SYSTEM Distributed_Control_System_OPCUA_4Diac
  (* Version 1.0, Author, Eclipse 4diac *)
  APPLICATION Distributed_Control_System_OPCUA_4DiacApp
    FBS
      HMI_COME_TO_ME : HMI_COME_TO_ME;
      EMERGENCY_STOP : RADIO_BOOL(QI := 1, LABEL1 := Start, LABEL0 := Emergency STOP, IN := 0);
      INPUT_BOX : IN_ANY(QI := 1, W := 20, TYPE := INT);
      COME_TO_ME : RADIO_BOOL(QI := 1, LABEL1 := Come to me, LABEL0 := STOP, IN := 0);
      FOLLOW_ME : RADIO_BOOL(QI := 1, LABEL1 := Follow me, LABEL0 := STOP, IN := 0);
      FOLLOW_MACHINE : RADIO_BOOL(QI := 1, LABEL1 := Follow machine, LABEL0 := STOP, IN := 0);
      INT2INT : INT2INT;
      HMI_FOLLOW_ME : HMI_FOLLOW_ME;
      HMI_FOLLOW_MACHINE : HMI_FOLLOW_MACHINE;
      CRANE2_COME_TO_ME : CRANE2_COME_TO_ME;
      CRANE1_COME_TO_ME : CRANE1_COME_TO_ME;
      CRANE2_FOLLOW_ME : CRANE2_FOLLOW_ME;
      CRANE1_FOLLOW_MACHINE : CRANE1_FOLLOW_MACHINE;
      CRANE2_FOLLOW_MACHINE : CRANE2_FOLLOW_MACHINE;
      MASTER_SLAVE : RADIO_BOOL(QI := 1, LABEL1 := Activate Bridge, LABEL0 := Stop, IN := 0);
      ACTIVATE_TROLLEY : RADIO_BOOL(QI := 1, LABEL1 := Activate Trolley, LABEL0 := Stop, IN := 0);
      ACTIVATE_HOOK : RADIO_BOOL(QI := 1, LABEL1 := Hook Up, LABEL0 := Stop, IN := 0);
      CRANE_NR : RADIO_BOOL(QI := 1, LABEL1 := Select Crane Nr, LABEL0 := No, IN := 0);
      HOOK_UP_DOWN : RADIO_BOOL(QI := 1, LABEL1 := Hook Down, LABEL0 := Stop, IN := 0);
      SENSORS_ACTUATORS_2 : SENSORS_ACTUATORS;
      SENSORS_ACTUATORS_1 : SENSORS_ACTUATORS;
      CHOOSE_X : RADIO_BOOL(QI := 1, LABEL1 := Choose X, LABEL0 := No, IN := 0);
      CHOOSE_Y : RADIO_BOOL(QI := 1, LABEL1 := Choose Y, LABEL0 := No, IN := 0);
      BOOL2BOOL : BOOL2BOOL;
      BOOL2BOOL_1 : BOOL2BOOL;
      CRANE_1 : CLIENT_6_0(QI := 1, ID := opc_ua[opc.tcp://%CRANE1_IP%:4840#/Objects/1:CRANE1/SERVER1]);
      CEANE_2 : CLIENT_6_0(QI := 1, ID := opc_ua[opc.tcp://%CRANE2_IP%:4840#/Objects/1:CRANE2/SERVER2]);
      TYPE_CONVERTER : TYPE_CONVERTER_1I_11B;
      SERVER1 : SERVER_0_6(QI := 1, ID := opc_ua[/Objects/1:CRANE1]);
      FUNCTIONALITY_CONTROLLER : FUNCTIONALITY_CONTROLLER;
      CRANE_SELECTOR : CRANE_SELECTOR;
      FME_FMA_DECIDER : FME_FMA_DECIDER;
      CRANE1_FOLLOW_ME : CRANE1_FOLLOW_ME;
      SUBSCRIBE_10_2 : SUBSCRIBE_10(QI := 1, ID := 239.0.0.2:61497);
      SERVER2 : SERVER_0_6(QI := 1, ID := opc_ua[/Objects/1:CRANE2]);
      PUBLISH_10 : PUBLISH_10(QI := 1, ID := 239.0.0.2:61497);
      SUB1 : SUBSCRIBE_10(QI := 1, ID := 239.0.0.2:61497);
      PUBLISH_12 : PUBLISH_12(QI := 1, ID := 239.0.0.1:61496);
      SUBSCRIBE_12 : SUBSCRIBE_12(QI := 1, ID := 239.0.0.1:61496);
      START_STOP_CONTROLLER_1 : START_STOP_CONTROLLER;
      START_STOP_CONTROLLER_2 : START_STOP_CONTROLLER;
      REQUEST : DISPLAY_LOCAL_TIME;
      RESPONSE : DISPLAY_LOCAL_TIME;
      PERMITTER_2 : PERMITTER;
      PERMITTER_1 : PERMITTER;
      BOOL2BOOL_2 : BOOL2BOOL;
      BOOL2BOOL_3 : BOOL2BOOL;
    END_FBS
    EVENT_CONNECTIONS
      INPUT_BOX.IND TO INT2INT.REQ;
      EMERGENCY_STOP.INITO TO INPUT_BOX.INIT;
      INPUT_BOX.INITO TO COME_TO_ME.INIT;
      COME_TO_ME.INITO TO FOLLOW_ME.INIT;
      FOLLOW_ME.INITO TO FOLLOW_MACHINE.INIT;
      MASTER_SLAVE.INITO TO ACTIVATE_TROLLEY.INIT;
      ACTIVATE_TROLLEY.INITO TO ACTIVATE_HOOK.INIT;
      CRANE2_COME_TO_ME.CNF TO SENSORS_ACTUATORS_2.REQ;
      CRANE1_COME_TO_ME.CNF TO SENSORS_ACTUATORS_1.REQ;
      CRANE1_FOLLOW_MACHINE.CNF TO SENSORS_ACTUATORS_1.REQ;
      CHOOSE_X.INITO TO CHOOSE_Y.INIT;
      HOOK_UP_DOWN.INITO TO CHOOSE_X.INIT;
      CHOOSE_Y.IND TO BOOL2BOOL_1.REQ;
      CHOOSE_X.IND TO BOOL2BOOL.REQ;
      FOLLOW_MACHINE.INITO TO CRANE_NR.INIT;
      CRANE_NR.INITO TO MASTER_SLAVE.INIT;
      ACTIVATE_HOOK.INITO TO HOOK_UP_DOWN.INIT;
      SERVER1.IND TO CRANE1_COME_TO_ME.REQ;
      SERVER1.IND TO CRANE1_FOLLOW_MACHINE.REQ;
      SERVER1.INITO TO SENSORS_ACTUATORS_1.INIT;
      TYPE_CONVERTER.CNF TO HMI_COME_TO_ME.REQ;
      TYPE_CONVERTER.CNF TO HMI_FOLLOW_ME.REQ;
      TYPE_CONVERTER.CNF TO HMI_FOLLOW_MACHINE.REQ;
      TYPE_CONVERTER.CNF TO FUNCTIONALITY_CONTROLLER.TRIGGER;
      FUNCTIONALITY_CONTROLLER.CTM_OUT TO HMI_COME_TO_ME.TRIGGER_IN;
      SERVER1.IND TO SERVER1.RSP;
      CRANE2_FOLLOW_ME.CNF TO SENSORS_ACTUATORS_2.REQ;
      CRANE2_FOLLOW_MACHINE.CNF TO SENSORS_ACTUATORS_2.REQ;
      FUNCTIONALITY_CONTROLLER.FME_OUT TO HMI_FOLLOW_ME.TRIGGER_IN;
      FUNCTIONALITY_CONTROLLER.FMA_OUT TO HMI_FOLLOW_MACHINE.TRIGGER_IN;
      HMI_COME_TO_ME.TRIGGER_OUT TO CRANE_SELECTOR.CTM;
      HMI_FOLLOW_ME.TRIGGER_OUT TO CRANE_SELECTOR.FME;
      TYPE_CONVERTER.CNF TO CRANE_SELECTOR.REQ;
      HMI_FOLLOW_MACHINE.TRIGGER_OUT TO CRANE_SELECTOR.FMA;
      SENSORS_ACTUATORS_1.S_A_E TO CRANE1_COME_TO_ME.MPS_E;
      SENSORS_ACTUATORS_1.S_A_E TO CRANE1_FOLLOW_MACHINE.MPS_E;
      SENSORS_ACTUATORS_2.S_A_E TO CRANE2_FOLLOW_ME.MPS_E;
      SENSORS_ACTUATORS_2.S_A_E TO CRANE2_COME_TO_ME.MPS_E;
      SENSORS_ACTUATORS_2.S_A_E TO CRANE2_FOLLOW_MACHINE.MPS_E;
      HMI_COME_TO_ME.UPDATER_OUT TO HMI_FOLLOW_ME.REQ;
      HMI_COME_TO_ME.UPDATER_OUT TO HMI_FOLLOW_MACHINE.REQ;
      HMI_FOLLOW_ME.TRIGGER_OUT TO FME_FMA_DECIDER.FME_TRIGGER;
      HMI_FOLLOW_MACHINE.TRIGGER_OUT TO FME_FMA_DECIDER.FMA_TRIGGER;
      FME_FMA_DECIDER.TRIGGER TO HMI_COME_TO_ME.UPDATER_IN;
      CRANE1_FOLLOW_ME.CNF TO SENSORS_ACTUATORS_1.REQ;
      SENSORS_ACTUATORS_1.S_A_E TO CRANE1_FOLLOW_ME.MPS_E;
      SERVER1.IND TO CRANE1_FOLLOW_ME.REQ;
      SERVER2.INITO TO SUBSCRIBE_10_2.INIT;
      TYPE_CONVERTER.CNF TO PUBLISH_10.REQ;
      SERVER1.INITO TO SUB1.INIT;
      SUB1.IND TO CRANE1_COME_TO_ME.REQ;
      SUB1.IND TO CRANE1_FOLLOW_ME.REQ;
      SUB1.IND TO SENSORS_ACTUATORS_1.REQ;
      PUBLISH_12.INITO TO EMERGENCY_STOP.INIT;
      EMERGENCY_STOP.IND TO PUBLISH_12.REQ;
      INT2INT.CNF TO PUBLISH_12.REQ;
      COME_TO_ME.IND TO PUBLISH_12.REQ;
      FOLLOW_ME.IND TO PUBLISH_12.REQ;
      FOLLOW_MACHINE.IND TO PUBLISH_12.REQ;
      CRANE_NR.IND TO PUBLISH_12.REQ;
      MASTER_SLAVE.IND TO PUBLISH_12.REQ;
      ACTIVATE_TROLLEY.IND TO PUBLISH_12.REQ;
      ACTIVATE_HOOK.IND TO PUBLISH_12.REQ;
      HOOK_UP_DOWN.IND TO PUBLISH_12.REQ;
      BOOL2BOOL.CNF TO PUBLISH_12.REQ;
      BOOL2BOOL_1.CNF TO PUBLISH_12.REQ;
      SUBSCRIBE_12.IND TO TYPE_CONVERTER.REQ;
      SUBSCRIBE_12.INITO TO PUBLISH_10.INIT;
      SUBSCRIBE_12.INITO TO CRANE_1.INIT;
      SUBSCRIBE_12.INITO TO CEANE_2.INIT;
      SUB1.IND TO START_STOP_CONTROLLER_1.REQ;
      SUB1.INITO TO START_STOP_CONTROLLER_1.INIT;
      START_STOP_CONTROLLER_1.CNF TO CRANE1_FOLLOW_ME.REQ;
      START_STOP_CONTROLLER_1.CNF TO CRANE1_COME_TO_ME.REQ;
      START_STOP_CONTROLLER_2.CNF TO CRANE2_COME_TO_ME.REQ;
      START_STOP_CONTROLLER_2.CNF TO CRANE2_FOLLOW_MACHINE.REQ;
      START_STOP_CONTROLLER_2.CNF TO CRANE2_FOLLOW_ME.REQ;
      START_STOP_CONTROLLER_1.CNF TO CRANE1_FOLLOW_MACHINE.REQ;
      SUB1.IND TO CRANE1_FOLLOW_MACHINE.REQ;
      SERVER2.IND TO CRANE2_COME_TO_ME.REQ;
      SERVER2.IND TO CRANE2_FOLLOW_ME.REQ;
      SERVER2.IND TO CRANE2_FOLLOW_MACHINE.REQ;
      SERVER2.IND TO SERVER2.RSP;
      SUBSCRIBE_10_2.INITO TO SENSORS_ACTUATORS_2.INIT;
      SUBSCRIBE_10_2.INITO TO START_STOP_CONTROLLER_2.INIT;
      SUBSCRIBE_10_2.IND TO CRANE2_COME_TO_ME.REQ;
      SUBSCRIBE_10_2.IND TO CRANE2_FOLLOW_ME.REQ;
      SUBSCRIBE_10_2.IND TO CRANE2_FOLLOW_MACHINE.REQ;
      SUBSCRIBE_10_2.IND TO SENSORS_ACTUATORS_2.REQ;
      SUBSCRIBE_10_2.IND TO START_STOP_CONTROLLER_2.REQ;
      CRANE_SELECTOR.C2 TO CEANE_2.REQ;
      CRANE_SELECTOR.C1 TO CRANE_1.REQ;
      CRANE_1.CNF TO RESPONSE.REQ;
      CEANE_2.CNF TO RESPONSE.REQ;
      CRANE_SELECTOR.C1 TO REQUEST.REQ;
      CRANE_SELECTOR.C2 TO REQUEST.REQ;
      START_STOP_CONTROLLER_1.CNF TO PERMITTER_1.REQ;
      SENSORS_ACTUATORS_1.S_A_E TO PERMITTER_1.TRIGGER_IN;
      PERMITTER_1.TRIGGER_OUT TO CRANE1_FOLLOW_MACHINE.REQ;
      START_STOP_CONTROLLER_2.CNF TO PERMITTER_2.REQ;
      SENSORS_ACTUATORS_2.S_A_E TO PERMITTER_2.TRIGGER_IN;
      PERMITTER_2.TRIGGER_OUT TO CRANE2_FOLLOW_MACHINE.REQ;
    END_CONNECTIONS
    DATA_CONNECTIONS
      INPUT_BOX.OUT TO INT2INT.IN;
      SENSORS_ACTUATORS_2.CRANE_DIS_S TO CRANE2_COME_TO_ME.CRANE_DIS_S;
      SENSORS_ACTUATORS_1.CRANE_DIS_S TO CRANE1_COME_TO_ME.CRANE_DIS_S;
      SENSORS_ACTUATORS_1.CRANE_DIS_S TO CRANE1_FOLLOW_MACHINE.CRANE_DIS_S;
      SENSORS_ACTUATORS_2.CRANE_DIS_S TO CRANE2_FOLLOW_ME.CRANE_DIS_S;
      SENSORS_ACTUATORS_2.CRANE_DIS_S TO CRANE2_FOLLOW_MACHINE.CRANE_DIS_S;
      CHOOSE_Y.OUT TO BOOL2BOOL_1.IN;
      CHOOSE_X.OUT TO BOOL2BOOL.IN;
      TYPE_CONVERTER.BOOL11OUT TO HMI_COME_TO_ME.Choose_X;
      TYPE_CONVERTER.BOOL12OUT TO HMI_COME_TO_ME.Choose_Y;
      TYPE_CONVERTER.BOOL11OUT TO HMI_FOLLOW_ME.Choose_X;
      TYPE_CONVERTER.BOOL12OUT TO HMI_FOLLOW_ME.Choose_Y;
      TYPE_CONVERTER.BOOL12OUT TO HMI_FOLLOW_MACHINE.Choose_Y;
      HMI_COME_TO_ME.Output_X TO CRANE_SELECTOR.CTM_X_I;
      HMI_COME_TO_ME.Output_Y TO CRANE_SELECTOR.CTM_Y_I;
      HMI_FOLLOW_ME.Output_X TO CRANE_SELECTOR.FME_X_I;
      HMI_FOLLOW_ME.Output_Y TO CRANE_SELECTOR.FME_Y_I;
      HMI_FOLLOW_MACHINE.Output_X TO CRANE_SELECTOR.FMA_X_I;
      HMI_FOLLOW_MACHINE.Output_Y TO CRANE_SELECTOR.FMA_Y_I;
      SENSORS_ACTUATORS_1.HOOK_P TO CRANE1_COME_TO_ME.HOOK_P;
      SENSORS_ACTUATORS_1.BRIDGE_P TO CRANE1_COME_TO_ME.BRIDGE_P;
      SENSORS_ACTUATORS_1.TROLLEY_P TO CRANE1_COME_TO_ME.TROLLEY_P;
      CRANE1_COME_TO_ME.BRIDGE_F TO SENSORS_ACTUATORS_1.CTM_BRIDGE_F_I;
      CRANE1_COME_TO_ME.BRIDGE_B TO SENSORS_ACTUATORS_1.CTM_BRIGDE_B_I;
      CRANE1_COME_TO_ME.TROLLEY_F TO SENSORS_ACTUATORS_1.CTM_TROLLEY_F_I;
      CRANE1_COME_TO_ME.TROLLEY_B TO SENSORS_ACTUATORS_1.CTM_TROLLEY_B_I;
      CRANE1_COME_TO_ME.HOOK_U TO SENSORS_ACTUATORS_1.CTM_HOOK_U_I;
      CRANE1_COME_TO_ME.HOOK_D TO SENSORS_ACTUATORS_1.CTM_HOOK_D_I;
      SENSORS_ACTUATORS_1.BRIDGE_P TO CRANE1_FOLLOW_MACHINE.BRIDGE_P;
      SENSORS_ACTUATORS_1.TROLLEY_P TO CRANE1_FOLLOW_MACHINE.TROLLEY_P;
      SENSORS_ACTUATORS_1.HOOK_P TO CRANE1_FOLLOW_MACHINE.HOOK_P;
      CRANE1_FOLLOW_MACHINE.A_D_MPS TO SENSORS_ACTUATORS_1.FMA_ACTIVATE_MP;
      CRANE1_FOLLOW_MACHINE.BRIDGE_F TO SENSORS_ACTUATORS_1.FMA_BRIDGE_F_I;
      CRANE1_FOLLOW_MACHINE.BRIDGE_B TO SENSORS_ACTUATORS_1.FMA_BRIGDE_B_I;
      CRANE1_FOLLOW_MACHINE.TROLLEY_F TO SENSORS_ACTUATORS_1.FMA_TROLLEY_F_I;
      CRANE1_FOLLOW_MACHINE.TROLLEY_B TO SENSORS_ACTUATORS_1.FMA_TROLLEY_B_I;
      CRANE1_FOLLOW_MACHINE.HOOK_U TO SENSORS_ACTUATORS_1.FMA_HOOK_U_I;
      CRANE1_FOLLOW_MACHINE.HOOK_D TO SENSORS_ACTUATORS_1.FMA_HOOK_D_I;
      CRANE1_COME_TO_ME.A_D_MPS TO SENSORS_ACTUATORS_1.CTM_ACTIVATE_MP;
      SENSORS_ACTUATORS_2.HOOK_P TO CRANE2_COME_TO_ME.HOOK_P;
      SENSORS_ACTUATORS_2.TROLLEY_P TO CRANE2_COME_TO_ME.TROLLEY_P;
      SENSORS_ACTUATORS_2.BRIDGE_P TO CRANE2_COME_TO_ME.BRIDGE_P;
      SENSORS_ACTUATORS_2.BRIDGE_P TO CRANE2_FOLLOW_ME.BRIDGE_P;
      SENSORS_ACTUATORS_2.BRIDGE_P TO CRANE2_FOLLOW_MACHINE.BRIDGE_P;
      SENSORS_ACTUATORS_2.TROLLEY_P TO CRANE2_FOLLOW_ME.TROLLEY_P;
      SENSORS_ACTUATORS_2.TROLLEY_P TO CRANE2_FOLLOW_MACHINE.TROLLEY_P;
      SENSORS_ACTUATORS_2.HOOK_P TO CRANE2_FOLLOW_ME.HOOK_P;
      SENSORS_ACTUATORS_2.HOOK_P TO CRANE2_FOLLOW_MACHINE.HOOK_P;
      CRANE2_COME_TO_ME.A_D_MPS TO SENSORS_ACTUATORS_2.CTM_ACTIVATE_MP;
      CRANE2_COME_TO_ME.BRIDGE_F TO SENSORS_ACTUATORS_2.CTM_BRIDGE_F_I;
      CRANE2_COME_TO_ME.BRIDGE_B TO SENSORS_ACTUATORS_2.CTM_BRIGDE_B_I;
      CRANE2_COME_TO_ME.TROLLEY_F TO SENSORS_ACTUATORS_2.CTM_TROLLEY_F_I;
      CRANE2_COME_TO_ME.TROLLEY_B TO SENSORS_ACTUATORS_2.CTM_TROLLEY_B_I;
      CRANE2_COME_TO_ME.HOOK_U TO SENSORS_ACTUATORS_2.CTM_HOOK_U_I;
      CRANE2_COME_TO_ME.HOOK_D TO SENSORS_ACTUATORS_2.CTM_HOOK_D_I;
      CRANE2_FOLLOW_ME.A_D_MPS TO SENSORS_ACTUATORS_2.FME_ACTIVATE_MP;
      CRANE2_FOLLOW_ME.BRIDGE_F TO SENSORS_ACTUATORS_2.FME_BRIDGE_F_I;
      CRANE2_FOLLOW_ME.BRIDGE_B TO SENSORS_ACTUATORS_2.FME_BRIGDE_B_I;
      CRANE2_FOLLOW_ME.TROLLEY_F TO SENSORS_ACTUATORS_2.FME_TROLLEY_F_I;
      CRANE2_FOLLOW_ME.TROLLEY_B TO SENSORS_ACTUATORS_2.FME_TROLLEY_B_I;
      CRANE2_FOLLOW_ME.HOOK_U TO SENSORS_ACTUATORS_2.FME_HOOK_U_I;
      CRANE2_FOLLOW_ME.HOOK_D TO SENSORS_ACTUATORS_2.FME_HOOK_D_I;
      CRANE2_FOLLOW_MACHINE.A_D_MPS TO SENSORS_ACTUATORS_2.FMA_ACTIVATE_MP;
      CRANE2_FOLLOW_MACHINE.BRIDGE_F TO SENSORS_ACTUATORS_2.FMA_BRIDGE_F_I;
      CRANE2_FOLLOW_MACHINE.BRIDGE_B TO SENSORS_ACTUATORS_2.FMA_BRIGDE_B_I;
      CRANE2_FOLLOW_MACHINE.TROLLEY_F TO SENSORS_ACTUATORS_2.FMA_TROLLEY_F_I;
      CRANE2_FOLLOW_MACHINE.TROLLEY_B TO SENSORS_ACTUATORS_2.FMA_TROLLEY_B_I;
      CRANE2_FOLLOW_MACHINE.HOOK_U TO SENSORS_ACTUATORS_2.FMA_HOOK_U_I;
      CRANE2_FOLLOW_MACHINE.HOOK_D TO SENSORS_ACTUATORS_2.FMA_HOOK_D_I;
      HMI_COME_TO_ME.Output_X TO HMI_FOLLOW_ME.CTM_X;
      HMI_COME_TO_ME.Output_Y TO HMI_FOLLOW_ME.CTM_Y;
      HMI_COME_TO_ME.Output_X TO HMI_FOLLOW_MACHINE.CTM_X;
      HMI_COME_TO_ME.Output_Y TO HMI_FOLLOW_MACHINE.CTM_Y;
      HMI_FOLLOW_ME.Output_X TO FME_FMA_DECIDER.X_FME;
      HMI_FOLLOW_ME.Output_Y TO FME_FMA_DECIDER.Y_FME;
      HMI_FOLLOW_MACHINE.Output_X TO FME_FMA_DECIDER.X_FMA;
      HMI_FOLLOW_MACHINE.Output_Y TO FME_FMA_DECIDER.Y_FMA;
      FME_FMA_DECIDER.X_FME_FMA TO HMI_COME_TO_ME.FME_FMA_X;
      FME_FMA_DECIDER.Y_FME_FMA TO HMI_COME_TO_ME.FME_FMA_Y;
      CRANE_SELECTOR.CTM_X_1 TO CRANE_1.SD_1;
      CRANE_SELECTOR.CTM_Y_1 TO CRANE_1.SD_2;
      CRANE_SELECTOR.FME_X_1 TO CRANE_1.SD_3;
      CRANE_SELECTOR.FME_Y_1 TO CRANE_1.SD_4;
      CRANE_SELECTOR.FMA_X_1 TO CRANE_1.SD_5;
      CRANE_SELECTOR.FMA_Y_1 TO CRANE_1.SD_6;
      CRANE_SELECTOR.CTM_X_2 TO CEANE_2.SD_1;
      CRANE_SELECTOR.CTM_Y_2 TO CEANE_2.SD_2;
      CRANE_SELECTOR.FME_X_2 TO CEANE_2.SD_3;
      CRANE_SELECTOR.FME_Y_2 TO CEANE_2.SD_4;
      CRANE_SELECTOR.FMA_X_2 TO CEANE_2.SD_5;
      CRANE_SELECTOR.FMA_Y_2 TO CEANE_2.SD_6;
      CRANE1_FOLLOW_ME.HOOK_D TO SENSORS_ACTUATORS_1.FME_HOOK_D_I;
      CRANE1_FOLLOW_ME.HOOK_U TO SENSORS_ACTUATORS_1.FME_HOOK_U_I;
      CRANE1_FOLLOW_ME.TROLLEY_B TO SENSORS_ACTUATORS_1.FME_TROLLEY_B_I;
      CRANE1_FOLLOW_ME.TROLLEY_F TO SENSORS_ACTUATORS_1.FME_TROLLEY_F_I;
      CRANE1_FOLLOW_ME.BRIDGE_B TO SENSORS_ACTUATORS_1.FME_BRIGDE_B_I;
      CRANE1_FOLLOW_ME.BRIDGE_F TO SENSORS_ACTUATORS_1.FME_BRIDGE_F_I;
      CRANE1_FOLLOW_ME.A_D_MPS TO SENSORS_ACTUATORS_1.FME_ACTIVATE_MP;
      SENSORS_ACTUATORS_1.CRANE_DIS_S TO CRANE1_FOLLOW_ME.CRANE_DIS_S;
      SENSORS_ACTUATORS_1.HOOK_P TO CRANE1_FOLLOW_ME.HOOK_P;
      SENSORS_ACTUATORS_1.TROLLEY_P TO CRANE1_FOLLOW_ME.TROLLEY_P;
      SENSORS_ACTUATORS_1.BRIDGE_P TO CRANE1_FOLLOW_ME.BRIDGE_P;
      SUBSCRIBE_10_2.RD_1 TO CRANE2_COME_TO_ME.E_STOP;
      SUBSCRIBE_10_2.RD_1 TO CRANE2_FOLLOW_ME.E_STOP;
      SUBSCRIBE_10_2.RD_1 TO CRANE2_FOLLOW_MACHINE.E_STOP;
      SUBSCRIBE_10_2.RD_2 TO CRANE2_COME_TO_ME.TEXT_BOX;
      SUBSCRIBE_10_2.RD_2 TO CRANE2_FOLLOW_ME.TEXT_BOX;
      SUBSCRIBE_10_2.RD_2 TO CRANE2_FOLLOW_MACHINE.TEXT_BOX;
      SUBSCRIBE_10_2.RD_6 TO CRANE2_COME_TO_ME.CHOOSE_CRANE;
      SUBSCRIBE_10_2.RD_6 TO CRANE2_FOLLOW_ME.CHOOSE_CRANE;
      SUBSCRIBE_10_2.RD_6 TO CRANE2_FOLLOW_MACHINE.CHOOSE_CRANE;
      SUBSCRIBE_10_2.RD_8 TO CRANE2_COME_TO_ME.ACTIVATE_TROLLEY;
      SUBSCRIBE_10_2.RD_8 TO CRANE2_FOLLOW_ME.ACTIVATE_TROLLEY;
      SUBSCRIBE_10_2.RD_8 TO CRANE2_FOLLOW_MACHINE.ACTIVATE_TROLLEY;
      SUBSCRIBE_10_2.RD_9 TO CRANE2_COME_TO_ME.HOOK_U_IN;
      SUBSCRIBE_10_2.RD_9 TO CRANE2_FOLLOW_ME.HOOK_U_IN;
      SUBSCRIBE_10_2.RD_9 TO CRANE2_FOLLOW_MACHINE.HOOK_U_IN;
      SUBSCRIBE_10_2.RD_10 TO CRANE2_COME_TO_ME.HOOK_D_IN;
      SUBSCRIBE_10_2.RD_10 TO CRANE2_FOLLOW_ME.HOOK_D_IN;
      SUBSCRIBE_10_2.RD_10 TO CRANE2_FOLLOW_MACHINE.HOOK_D_IN;
      SERVER2.RD_1 TO CRANE2_COME_TO_ME.X_B_LOC;
      SERVER2.RD_2 TO CRANE2_COME_TO_ME.Y_T_LOC;
      SERVER2.RD_3 TO CRANE2_FOLLOW_ME.X_B_LOC;
      SERVER2.RD_4 TO CRANE2_FOLLOW_ME.Y_T_LOC;
      SERVER2.RD_5 TO CRANE2_FOLLOW_MACHINE.X_B_LOC;
      SERVER2.RD_6 TO CRANE2_FOLLOW_MACHINE.Y_T_LOC;
      SUBSCRIBE_10_2.RD_1 TO SENSORS_ACTUATORS_2.E_STOP;
      SERVER1.RD_1 TO CRANE1_COME_TO_ME.X_B_LOC;
      SERVER1.RD_2 TO CRANE1_COME_TO_ME.Y_T_LOC;
      SERVER1.RD_3 TO CRANE1_FOLLOW_ME.X_B_LOC;
      SERVER1.RD_4 TO CRANE1_FOLLOW_ME.Y_T_LOC;
      SERVER1.RD_5 TO CRANE1_FOLLOW_MACHINE.X_B_LOC;
      SERVER1.RD_6 TO CRANE1_FOLLOW_MACHINE.Y_T_LOC;
      TYPE_CONVERTER.BOOL11OUT TO HMI_FOLLOW_MACHINE.Choose_X;
      TYPE_CONVERTER.BOOL1OUT TO PUBLISH_10.SD_1;
      TYPE_CONVERTER.INT2OUT TO PUBLISH_10.SD_2;
      TYPE_CONVERTER.BOOL3OUT TO PUBLISH_10.SD_3;
      TYPE_CONVERTER.BOOL4OUT TO PUBLISH_10.SD_4;
      TYPE_CONVERTER.BOOL5OUT TO PUBLISH_10.SD_5;
      TYPE_CONVERTER.BOOL6OUT TO PUBLISH_10.SD_6;
      TYPE_CONVERTER.BOOL7OUT TO PUBLISH_10.SD_7;
      TYPE_CONVERTER.BOOL8OUT TO PUBLISH_10.SD_8;
      TYPE_CONVERTER.BOOL9OUT TO PUBLISH_10.SD_9;
      TYPE_CONVERTER.BOOL10OUT TO PUBLISH_10.SD_10;
      SUB1.RD_1 TO CRANE1_COME_TO_ME.E_STOP;
      SUB1.RD_1 TO CRANE1_FOLLOW_ME.E_STOP;
      SUB1.RD_1 TO CRANE1_FOLLOW_MACHINE.E_STOP;
      SUB1.RD_1 TO SENSORS_ACTUATORS_1.E_STOP;
      SUB1.RD_2 TO CRANE1_COME_TO_ME.TEXT_BOX;
      SUB1.RD_2 TO CRANE1_FOLLOW_ME.TEXT_BOX;
      SUB1.RD_2 TO CRANE1_FOLLOW_MACHINE.TEXT_BOX;
      SUB1.RD_6 TO CRANE1_COME_TO_ME.CHOOSE_CRANE;
      SUB1.RD_6 TO CRANE1_FOLLOW_ME.CHOOSE_CRANE;
      SUB1.RD_6 TO CRANE1_FOLLOW_MACHINE.CHOOSE_CRANE;
      SUB1.RD_8 TO CRANE1_COME_TO_ME.ACTIVATE_TROLLEY;
      SUB1.RD_8 TO CRANE1_FOLLOW_ME.ACTIVATE_TROLLEY;
      SUB1.RD_8 TO CRANE1_FOLLOW_MACHINE.ACTIVATE_TROLLEY;
      SUB1.RD_9 TO CRANE1_COME_TO_ME.HOOK_U_IN;
      SUB1.RD_9 TO CRANE1_FOLLOW_ME.HOOK_U_IN;
      SUB1.RD_9 TO CRANE1_FOLLOW_MACHINE.HOOK_U_IN;
      SUB1.RD_10 TO CRANE1_COME_TO_ME.HOOK_D_IN;
      SUB1.RD_10 TO CRANE1_FOLLOW_ME.HOOK_D_IN;
      SUB1.RD_10 TO CRANE1_FOLLOW_MACHINE.HOOK_D_IN;
      EMERGENCY_STOP.OUT TO PUBLISH_12.SD_1;
      INT2INT.OUT TO PUBLISH_12.SD_2;
      COME_TO_ME.OUT TO PUBLISH_12.SD_3;
      FOLLOW_ME.OUT TO PUBLISH_12.SD_4;
      FOLLOW_MACHINE.OUT TO PUBLISH_12.SD_5;
      CRANE_NR.OUT TO PUBLISH_12.SD_6;
      MASTER_SLAVE.OUT TO PUBLISH_12.SD_7;
      ACTIVATE_TROLLEY.OUT TO PUBLISH_12.SD_8;
      ACTIVATE_HOOK.OUT TO PUBLISH_12.SD_9;
      HOOK_UP_DOWN.OUT TO PUBLISH_12.SD_10;
      BOOL2BOOL.OUT TO PUBLISH_12.SD_11;
      BOOL2BOOL_1.OUT TO PUBLISH_12.SD_12;
      SUBSCRIBE_12.RD_1 TO TYPE_CONVERTER.BOOL1IN;
      SUBSCRIBE_12.RD_2 TO TYPE_CONVERTER.INT2IN;
      SUBSCRIBE_12.RD_12 TO TYPE_CONVERTER.BOOL12IN;
      SUBSCRIBE_12.RD_11 TO TYPE_CONVERTER.BOOL11IN;
      SUBSCRIBE_12.RD_10 TO TYPE_CONVERTER.BOOL10IN;
      SUBSCRIBE_12.RD_9 TO TYPE_CONVERTER.BOOL9IN;
      SUBSCRIBE_12.RD_8 TO TYPE_CONVERTER.BOOL8IN;
      SUBSCRIBE_12.RD_7 TO TYPE_CONVERTER.BOOL7IN;
      SUBSCRIBE_12.RD_6 TO TYPE_CONVERTER.BOOL6IN;
      SUBSCRIBE_12.RD_5 TO TYPE_CONVERTER.BOOL5IN;
      SUBSCRIBE_12.RD_4 TO TYPE_CONVERTER.BOOL4IN;
      SUBSCRIBE_12.RD_3 TO TYPE_CONVERTER.BOOL3IN;
      TYPE_CONVERTER.INT2OUT TO CRANE_SELECTOR.Text_box;
      TYPE_CONVERTER.BOOL6OUT TO CRANE_SELECTOR.choose_crane;
      TYPE_CONVERTER.BOOL1OUT TO HMI_COME_TO_ME.E_Stop;
      TYPE_CONVERTER.BOOL1OUT TO HMI_FOLLOW_ME.E_Stop;
      TYPE_CONVERTER.BOOL1OUT TO HMI_FOLLOW_MACHINE.E_Stop;
      TYPE_CONVERTER.INT2OUT TO HMI_COME_TO_ME.XY;
      TYPE_CONVERTER.INT2OUT TO HMI_FOLLOW_ME.XY;
      TYPE_CONVERTER.INT2OUT TO HMI_FOLLOW_MACHINE.XY;
      TYPE_CONVERTER.BOOL3OUT TO HMI_COME_TO_ME.N_Stop;
      TYPE_CONVERTER.BOOL1OUT TO FUNCTIONALITY_CONTROLLER.E_STOP;
      TYPE_CONVERTER.BOOL3OUT TO FUNCTIONALITY_CONTROLLER.CTM_N_IN;
      TYPE_CONVERTER.BOOL4OUT TO FUNCTIONALITY_CONTROLLER.FME_N_IN;
      TYPE_CONVERTER.BOOL5OUT TO FUNCTIONALITY_CONTROLLER.FMA_N_IN;
      TYPE_CONVERTER.BOOL4OUT TO HMI_FOLLOW_ME.N_Stop;
      TYPE_CONVERTER.BOOL5OUT TO HMI_FOLLOW_MACHINE.N_Stop;
      SUB1.RD_3 TO START_STOP_CONTROLLER_1.CTM;
      SUB1.RD_4 TO START_STOP_CONTROLLER_1.FME;
      SUB1.RD_5 TO START_STOP_CONTROLLER_1.FMA;
      START_STOP_CONTROLLER_1.CTM_O TO CRANE1_COME_TO_ME.N_STOP;
      START_STOP_CONTROLLER_1.FME_O TO CRANE1_FOLLOW_ME.N_STOP;
      START_STOP_CONTROLLER_1.FMA_O TO CRANE1_FOLLOW_MACHINE.N_STOP;
      SUBSCRIBE_10_2.RD_3 TO START_STOP_CONTROLLER_2.CTM;
      SUBSCRIBE_10_2.RD_4 TO START_STOP_CONTROLLER_2.FME;
      SUBSCRIBE_10_2.RD_5 TO START_STOP_CONTROLLER_2.FMA;
      START_STOP_CONTROLLER_2.CTM_O TO CRANE2_COME_TO_ME.N_STOP;
      START_STOP_CONTROLLER_2.FME_O TO CRANE2_FOLLOW_ME.N_STOP;
      START_STOP_CONTROLLER_2.FMA_O TO CRANE2_FOLLOW_MACHINE.N_STOP;
      START_STOP_CONTROLLER_1.FMA_O TO PERMITTER_1.N_STOP;
      SUB1.RD_1 TO PERMITTER_1.E_STOP;
      START_STOP_CONTROLLER_2.FMA_O TO PERMITTER_2.N_STOP;
      SUBSCRIBE_10_2.RD_1 TO PERMITTER_2.E_STOP;
      BOOL2BOOL_2.OUT TO BOOL2BOOL_2.IN;
      SUB1.RD_7 TO CRANE1_COME_TO_ME.ACTIVATE_BRIDGE;
      SUB1.RD_7 TO CRANE1_FOLLOW_MACHINE.ACTIVATE_BRIDGE;
      SUB1.RD_7 TO CRANE1_FOLLOW_ME.ACTIVATE_BRIDGE;
      SUBSCRIBE_10_2.RD_7 TO CRANE2_COME_TO_ME.ACTIVATE_BRIDGE;
      SUBSCRIBE_10_2.RD_7 TO CRANE2_FOLLOW_ME.ACTIVATE_BRIDGE;
      SUBSCRIBE_10_2.RD_7 TO CRANE2_FOLLOW_MACHINE.ACTIVATE_BRIDGE;
    END_CONNECTIONS
  END_APPLICATION
  DEVICE HMI_DEVICE : FORTE_PC(MGR_ID := "localhost:61497")
    {SET_ATTRIBUTE(Profile, HOLOBLOC)} (* device profile *)
    RESOURCE EMB_RES : EMB_RES
      FBS
        HMI_FOLLOW_ME : HMI_FOLLOW_ME;
        HMI_COME_TO_ME : HMI_COME_TO_ME;
        TYPE_CONVERTER : TYPE_CONVERTER_1I_11B;
        FUNCTIONALITY_CONTROLLER : FUNCTIONALITY_CONTROLLER;
        HMI_FOLLOW_MACHINE : HMI_FOLLOW_MACHINE;
        CRANE_1 : CLIENT_6_0(QI := 1, ID := opc_ua[opc.tcp://%CRANE1_IP%:4840#/Objects/1:CRANE1/SERVER1]);
        CEANE_2 : CLIENT_6_0(QI := 1, ID := opc_ua[opc.tcp://%CRANE2_IP%:4840#/Objects/1:CRANE2/SERVER2]);
        CRANE_SELECTOR : CRANE_SELECTOR;
        FME_FMA_DECIDER : FME_FMA_DECIDER;
        PUBLISH_10 : PUBLISH_10(QI := 1, ID := 239.0.0.2:61497);
        SUBSCRIBE_12 : SUBSCRIBE_12(QI := 1, ID := 239.0.0.1:61496);
        REQUEST : DISPLAY_LOCAL_TIME;
        RESPONSE : DISPLAY_LOCAL_TIME;
      END_FBS
      EVENT_CONNECTIONS
        TYPE_CONVERTER.CNF TO HMI_COME_TO_ME.REQ;
        TYPE_CONVERTER.CNF TO HMI_FOLLOW_ME.REQ;
        TYPE_CONVERTER.CNF TO FUNCTIONALITY_CONTROLLER.TRIGGER;
        FUNCTIONALITY_CONTROLLER.CTM_OUT TO HMI_COME_TO_ME.TRIGGER_IN;
        TYPE_CONVERTER.CNF TO HMI_FOLLOW_MACHINE.REQ;
        FUNCTIONALITY_CONTROLLER.FME_OUT TO HMI_FOLLOW_ME.TRIGGER_IN;
        FUNCTIONALITY_CONTROLLER.FMA_OUT TO HMI_FOLLOW_MACHINE.TRIGGER_IN;
        HMI_COME_TO_ME.TRIGGER_OUT TO CRANE_SELECTOR.CTM;
        HMI_FOLLOW_ME.TRIGGER_OUT TO CRANE_SELECTOR.FME;
        TYPE_CONVERTER.CNF TO CRANE_SELECTOR.REQ;
        HMI_FOLLOW_MACHINE.TRIGGER_OUT TO CRANE_SELECTOR.FMA;
        HMI_COME_TO_ME.UPDATER_OUT TO HMI_FOLLOW_ME.REQ;
        HMI_COME_TO_ME.UPDATER_OUT TO HMI_FOLLOW_MACHINE.REQ;
        HMI_FOLLOW_ME.TRIGGER_OUT TO FME_FMA_DECIDER.FME_TRIGGER;
        HMI_FOLLOW_MACHINE.TRIGGER_OUT TO FME_FMA_DECIDER.FMA_TRIGGER;
        FME_FMA_DECIDER.TRIGGER TO HMI_COME_TO_ME.UPDATER_IN;
        TYPE_CONVERTER.CNF TO PUBLISH_10.REQ;
        SUBSCRIBE_12.IND TO TYPE_CONVERTER.REQ;
        SUBSCRIBE_12.INITO TO PUBLISH_10.INIT;
        START.COLD TO SUBSCRIBE_12.INIT;
        START.WARM TO SUBSCRIBE_12.INIT;
        SUBSCRIBE_12.INITO TO CRANE_1.INIT;
        SUBSCRIBE_12.INITO TO CEANE_2.INIT;
        CRANE_SELECTOR.C2 TO CEANE_2.REQ;
        CRANE_SELECTOR.C1 TO CRANE_1.REQ;
        CRANE_1.CNF TO RESPONSE.REQ;
        CEANE_2.CNF TO RESPONSE.REQ;
        CRANE_SELECTOR.C1 TO REQUEST.REQ;
        CRANE_SELECTOR.C2 TO REQUEST.REQ;
      END_CONNECTIONS
      DATA_CONNECTIONS
        TYPE_CONVERTER.BOOL11OUT TO HMI_COME_TO_ME.Choose_X;
        TYPE_CONVERTER.BOOL11OUT TO HMI_FOLLOW_ME.Choose_X;
        TYPE_CONVERTER.BOOL12OUT TO HMI_COME_TO_ME.Choose_Y;
        TYPE_CONVERTER.BOOL12OUT TO HMI_FOLLOW_ME.Choose_Y;
        TYPE_CONVERTER.BOOL12OUT TO HMI_FOLLOW_MACHINE.Choose_Y;
        HMI_COME_TO_ME.Output_X TO CRANE_SELECTOR.CTM_X_I;
        HMI_COME_TO_ME.Output_Y TO CRANE_SELECTOR.CTM_Y_I;
        HMI_FOLLOW_ME.Output_X TO CRANE_SELECTOR.FME_X_I;
        HMI_FOLLOW_ME.Output_Y TO CRANE_SELECTOR.FME_Y_I;
        HMI_FOLLOW_MACHINE.Output_X TO CRANE_SELECTOR.FMA_X_I;
        HMI_FOLLOW_MACHINE.Output_Y TO CRANE_SELECTOR.FMA_Y_I;
        HMI_COME_TO_ME.Output_X TO HMI_FOLLOW_ME.CTM_X;
        HMI_COME_TO_ME.Output_Y TO HMI_FOLLOW_ME.CTM_Y;
        HMI_COME_TO_ME.Output_X TO HMI_FOLLOW_MACHINE.CTM_X;
        HMI_COME_TO_ME.Output_Y TO HMI_FOLLOW_MACHINE.CTM_Y;
        HMI_FOLLOW_ME.Output_X TO FME_FMA_DECIDER.X_FME;
        HMI_FOLLOW_ME.Output_Y TO FME_FMA_DECIDER.Y_FME;
        HMI_FOLLOW_MACHINE.Output_X TO FME_FMA_DECIDER.X_FMA;
        HMI_FOLLOW_MACHINE.Output_Y TO FME_FMA_DECIDER.Y_FMA;
        FME_FMA_DECIDER.X_FME_FMA TO HMI_COME_TO_ME.FME_FMA_X;
        FME_FMA_DECIDER.Y_FME_FMA TO HMI_COME_TO_ME.FME_FMA_Y;
        CRANE_SELECTOR.CTM_X_1 TO CRANE_1.SD_1;
        CRANE_SELECTOR.CTM_Y_1 TO CRANE_1.SD_2;
        CRANE_SELECTOR.FME_X_1 TO CRANE_1.SD_3;
        CRANE_SELECTOR.FME_Y_1 TO CRANE_1.SD_4;
        CRANE_SELECTOR.FMA_X_1 TO CRANE_1.SD_5;
        CRANE_SELECTOR.FMA_Y_1 TO CRANE_1.SD_6;
        CRANE_SELECTOR.CTM_X_2 TO CEANE_2.SD_1;
        CRANE_SELECTOR.CTM_Y_2 TO CEANE_2.SD_2;
        CRANE_SELECTOR.FME_X_2 TO CEANE_2.SD_3;
        CRANE_SELECTOR.FME_Y_2 TO CEANE_2.SD_4;
        CRANE_SELECTOR.FMA_X_2 TO CEANE_2.SD_5;
        CRANE_SELECTOR.FMA_Y_2 TO CEANE_2.SD_6;
        TYPE_CONVERTER.BOOL11OUT TO HMI_FOLLOW_MACHINE.Choose_X;
        TYPE_CONVERTER.BOOL1OUT TO PUBLISH_10.SD_1;
        TYPE_CONVERTER.INT2OUT TO PUBLISH_10.SD_2;
        TYPE_CONVERTER.BOOL3OUT TO PUBLISH_10.SD_3;
        TYPE_CONVERTER.BOOL4OUT TO PUBLISH_10.SD_4;
        TYPE_CONVERTER.BOOL5OUT TO PUBLISH_10.SD_5;
        TYPE_CONVERTER.BOOL6OUT TO PUBLISH_10.SD_6;
        TYPE_CONVERTER.BOOL7OUT TO PUBLISH_10.SD_7;
        TYPE_CONVERTER.BOOL8OUT TO PUBLISH_10.SD_8;
        TYPE_CONVERTER.BOOL9OUT TO PUBLISH_10.SD_9;
        TYPE_CONVERTER.BOOL10OUT TO PUBLISH_10.SD_10;
        SUBSCRIBE_12.RD_1 TO TYPE_CONVERTER.BOOL1IN;
        SUBSCRIBE_12.RD_2 TO TYPE_CONVERTER.INT2IN;
        SUBSCRIBE_12.RD_12 TO TYPE_CONVERTER.BOOL12IN;
        SUBSCRIBE_12.RD_11 TO TYPE_CONVERTER.BOOL11IN;
        SUBSCRIBE_12.RD_10 TO TYPE_CONVERTER.BOOL10IN;
        SUBSCRIBE_12.RD_9 TO TYPE_CONVERTER.BOOL9IN;
        SUBSCRIBE_12.RD_8 TO TYPE_CONVERTER.BOOL8IN;
        SUBSCRIBE_12.RD_7 TO TYPE_CONVERTER.BOOL7IN;
        SUBSCRIBE_12.RD_6 TO TYPE_CONVERTER.BOOL6IN;
        SUBSCRIBE_12.RD_5 TO TYPE_CONVERTER.BOOL5IN;
        SUBSCRIBE_12.RD_4 TO TYPE_CONVERTER.BOOL4IN;
        SUBSCRIBE_12.RD_3 TO TYPE_CONVERTER.BOOL3IN;
        TYPE_CONVERTER.INT2OUT TO CRANE_SELECTOR.Text_box;
        TYPE_CONVERTER.BOOL6OUT TO CRANE_SELECTOR.choose_crane;
        TYPE_CONVERTER.BOOL1OUT TO HMI_COME_TO_ME.E_Stop;
        TYPE_CONVERTER.BOOL1OUT TO HMI_FOLLOW_ME.E_Stop;
        TYPE_CONVERTER.BOOL1OUT TO HMI_FOLLOW_MACHINE.E_Stop;
        TYPE_CONVERTER.INT2OUT TO HMI_COME_TO_ME.XY;
        TYPE_CONVERTER.INT2OUT TO HMI_FOLLOW_ME.XY;
        TYPE_CONVERTER.INT2OUT TO HMI_FOLLOW_MACHINE.XY;
        TYPE_CONVERTER.BOOL3OUT TO HMI_COME_TO_ME.N_Stop;
        TYPE_CONVERTER.BOOL1OUT TO FUNCTIONALITY_CONTROLLER.E_STOP;
        TYPE_CONVERTER.BOOL3OUT TO FUNCTIONALITY_CONTROLLER.CTM_N_IN;
        TYPE_CONVERTER.BOOL4OUT TO FUNCTIONALITY_CONTROLLER.FME_N_IN;
        TYPE_CONVERTER.BOOL5OUT TO FUNCTIONALITY_CONTROLLER.FMA_N_IN;
        TYPE_CONVERTER.BOOL4OUT TO HMI_FOLLOW_ME.N_Stop;
        TYPE_CONVERTER.BOOL5OUT TO HMI_FOLLOW_MACHINE.N_Stop;
      END_CONNECTIONS
    END_RESOURCE
  END_DEVICE
  DEVICE CRANE_1_DEVICCE : FORTE_PC(MGR_ID := %CRANE1_IP%:61499)
    {SET_ATTRIBUTE(Profile, HOLOBLOC)} (* device profile *)
    RESOURCE EMB_RES : EMB_RES
      FBS
        CRANE1_COME_TO_ME : CRANE1_COME_TO_ME;
        CRANE1_FOLLOW_MACHINE : CRANE1_FOLLOW_MACHINE;
        CRANE1_FOLLOW_ME : CRANE1_FOLLOW_ME;
        SERVER1 : SERVER_0_6(QI := 1, ID := opc_ua[/Objects/1:CRANE1]);
        START_STOP_CONTROLLER_1 : START_STOP_CONTROLLER;
        SENSORS_ACTUATORS_1 : SENSORS_ACTUATORS;
        SUB1 : SUBSCRIBE_10(QI := 1, ID := 239.0.0.2:61497);
        PERMITTER_1 : PERMITTER;
      END_FBS
      EVENT_CONNECTIONS
        SERVER1.IND TO SERVER1.RSP;
        SERVER1.IND TO CRANE1_COME_TO_ME.REQ;
        SERVER1.IND TO CRANE1_FOLLOW_MACHINE.REQ;
        SERVER1.IND TO SERVER1.RSP;
        SERVER1.IND TO CRANE1_FOLLOW_ME.REQ;
        START_STOP_CONTROLLER_1.CNF TO CRANE1_FOLLOW_ME.REQ;
        START_STOP_CONTROLLER_1.CNF TO CRANE1_COME_TO_ME.REQ;
        START_STOP_CONTROLLER_1.CNF TO CRANE1_FOLLOW_MACHINE.REQ;
        CRANE1_COME_TO_ME.CNF TO SENSORS_ACTUATORS_1.REQ;
        CRANE1_FOLLOW_MACHINE.CNF TO SENSORS_ACTUATORS_1.REQ;
        CRANE1_FOLLOW_ME.CNF TO SENSORS_ACTUATORS_1.REQ;
        SERVER1.INITO TO SENSORS_ACTUATORS_1.INIT;
        SENSORS_ACTUATORS_1.S_A_E TO CRANE1_COME_TO_ME.MPS_E;
        SENSORS_ACTUATORS_1.S_A_E TO CRANE1_FOLLOW_MACHINE.MPS_E;
        SENSORS_ACTUATORS_1.S_A_E TO CRANE1_FOLLOW_ME.MPS_E;
        SERVER1.INITO TO SUB1.INIT;
        SUB1.INITO TO START_STOP_CONTROLLER_1.INIT;
        SUB1.IND TO CRANE1_COME_TO_ME.REQ;
        SUB1.IND TO CRANE1_FOLLOW_ME.REQ;
        SUB1.IND TO SENSORS_ACTUATORS_1.REQ;
        SUB1.IND TO START_STOP_CONTROLLER_1.REQ;
        SUB1.IND TO CRANE1_FOLLOW_MACHINE.REQ;
        START.COLD TO SERVER1.INIT;
        START.WARM TO SERVER1.INIT;
        SENSORS_ACTUATORS_1.S_A_E TO PERMITTER_1.TRIGGER_IN;
        START_STOP_CONTROLLER_1.CNF TO PERMITTER_1.REQ;
        PERMITTER_1.TRIGGER_OUT TO CRANE1_FOLLOW_MACHINE.REQ;
      END_CONNECTIONS
      DATA_CONNECTIONS
        SERVER1.RD_1 TO CRANE1_COME_TO_ME.X_B_LOC;
        SERVER1.RD_2 TO CRANE1_COME_TO_ME.Y_T_LOC;
        SERVER1.RD_3 TO CRANE1_FOLLOW_ME.X_B_LOC;
        SERVER1.RD_4 TO CRANE1_FOLLOW_ME.Y_T_LOC;
        SERVER1.RD_5 TO CRANE1_FOLLOW_MACHINE.X_B_LOC;
        SERVER1.RD_6 TO CRANE1_FOLLOW_MACHINE.Y_T_LOC;
        START_STOP_CONTROLLER_1.CTM_O TO CRANE1_COME_TO_ME.N_STOP;
        START_STOP_CONTROLLER_1.FME_O TO CRANE1_FOLLOW_ME.N_STOP;
        START_STOP_CONTROLLER_1.FMA_O TO CRANE1_FOLLOW_MACHINE.N_STOP;
        CRANE1_COME_TO_ME.A_D_MPS TO SENSORS_ACTUATORS_1.CTM_ACTIVATE_MP;
        CRANE1_COME_TO_ME.BRIDGE_F TO SENSORS_ACTUATORS_1.CTM_BRIDGE_F_I;
        CRANE1_COME_TO_ME.BRIDGE_B TO SENSORS_ACTUATORS_1.CTM_BRIGDE_B_I;
        CRANE1_COME_TO_ME.TROLLEY_F TO SENSORS_ACTUATORS_1.CTM_TROLLEY_F_I;
        CRANE1_COME_TO_ME.TROLLEY_B TO SENSORS_ACTUATORS_1.CTM_TROLLEY_B_I;
        CRANE1_COME_TO_ME.HOOK_U TO SENSORS_ACTUATORS_1.CTM_HOOK_U_I;
        CRANE1_COME_TO_ME.HOOK_D TO SENSORS_ACTUATORS_1.CTM_HOOK_D_I;
        CRANE1_FOLLOW_ME.A_D_MPS TO SENSORS_ACTUATORS_1.FME_ACTIVATE_MP;
        CRANE1_FOLLOW_ME.BRIDGE_F TO SENSORS_ACTUATORS_1.FME_BRIDGE_F_I;
        CRANE1_FOLLOW_ME.BRIDGE_B TO SENSORS_ACTUATORS_1.FME_BRIGDE_B_I;
        CRANE1_FOLLOW_ME.TROLLEY_F TO SENSORS_ACTUATORS_1.FME_TROLLEY_F_I;
        CRANE1_FOLLOW_ME.TROLLEY_B TO SENSORS_ACTUATORS_1.FME_TROLLEY_B_I;
        CRANE1_FOLLOW_ME.HOOK_U TO SENSORS_ACTUATORS_1.FME_HOOK_U_I;
        CRANE1_FOLLOW_ME.HOOK_D TO SENSORS_ACTUATORS_1.FME_HOOK_D_I;
        CRANE1_FOLLOW_MACHINE.A_D_MPS TO SENSORS_ACTUATORS_1.FMA_ACTIVATE_MP;
        CRANE1_FOLLOW_MACHINE.BRIDGE_F TO SENSORS_ACTUATORS_1.FMA_BRIDGE_F_I;
        CRANE1_FOLLOW_MACHINE.BRIDGE_B TO SENSORS_ACTUATORS_1.FMA_BRIGDE_B_I;
        CRANE1_FOLLOW_MACHINE.TROLLEY_F TO SENSORS_ACTUATORS_1.FMA_TROLLEY_F_I;
        CRANE1_FOLLOW_MACHINE.TROLLEY_B TO SENSORS_ACTUATORS_1.FMA_TROLLEY_B_I;
        CRANE1_FOLLOW_MACHINE.HOOK_U TO SENSORS_ACTUATORS_1.FMA_HOOK_U_I;
        CRANE1_FOLLOW_MACHINE.HOOK_D TO SENSORS_ACTUATORS_1.FMA_HOOK_D_I;
        SENSORS_ACTUATORS_1.BRIDGE_P TO CRANE1_COME_TO_ME.BRIDGE_P;
        SENSORS_ACTUATORS_1.BRIDGE_P TO CRANE1_FOLLOW_MACHINE.BRIDGE_P;
        SENSORS_ACTUATORS_1.BRIDGE_P TO CRANE1_FOLLOW_ME.BRIDGE_P;
        SENSORS_ACTUATORS_1.TROLLEY_P TO CRANE1_COME_TO_ME.TROLLEY_P;
        SENSORS_ACTUATORS_1.TROLLEY_P TO CRANE1_FOLLOW_MACHINE.TROLLEY_P;
        SENSORS_ACTUATORS_1.TROLLEY_P TO CRANE1_FOLLOW_ME.TROLLEY_P;
        SENSORS_ACTUATORS_1.HOOK_P TO CRANE1_COME_TO_ME.HOOK_P;
        SENSORS_ACTUATORS_1.HOOK_P TO CRANE1_FOLLOW_MACHINE.HOOK_P;
        SENSORS_ACTUATORS_1.HOOK_P TO CRANE1_FOLLOW_ME.HOOK_P;
        SENSORS_ACTUATORS_1.CRANE_DIS_S TO CRANE1_COME_TO_ME.CRANE_DIS_S;
        SENSORS_ACTUATORS_1.CRANE_DIS_S TO CRANE1_FOLLOW_MACHINE.CRANE_DIS_S;
        SENSORS_ACTUATORS_1.CRANE_DIS_S TO CRANE1_FOLLOW_ME.CRANE_DIS_S;
        SUB1.RD_1 TO CRANE1_COME_TO_ME.E_STOP;
        SUB1.RD_1 TO CRANE1_FOLLOW_ME.E_STOP;
        SUB1.RD_1 TO CRANE1_FOLLOW_MACHINE.E_STOP;
        SUB1.RD_1 TO SENSORS_ACTUATORS_1.E_STOP;
        SUB1.RD_2 TO CRANE1_COME_TO_ME.TEXT_BOX;
        SUB1.RD_2 TO CRANE1_FOLLOW_ME.TEXT_BOX;
        SUB1.RD_2 TO CRANE1_FOLLOW_MACHINE.TEXT_BOX;
        SUB1.RD_3 TO START_STOP_CONTROLLER_1.CTM;
        SUB1.RD_4 TO START_STOP_CONTROLLER_1.FME;
        SUB1.RD_5 TO START_STOP_CONTROLLER_1.FMA;
        SUB1.RD_6 TO CRANE1_COME_TO_ME.CHOOSE_CRANE;
        SUB1.RD_6 TO CRANE1_FOLLOW_ME.CHOOSE_CRANE;
        SUB1.RD_6 TO CRANE1_FOLLOW_MACHINE.CHOOSE_CRANE;
        SUB1.RD_8 TO CRANE1_COME_TO_ME.ACTIVATE_TROLLEY;
        SUB1.RD_8 TO CRANE1_FOLLOW_ME.ACTIVATE_TROLLEY;
        SUB1.RD_8 TO CRANE1_FOLLOW_MACHINE.ACTIVATE_TROLLEY;
        SUB1.RD_9 TO CRANE1_COME_TO_ME.HOOK_U_IN;
        SUB1.RD_9 TO CRANE1_FOLLOW_ME.HOOK_U_IN;
        SUB1.RD_9 TO CRANE1_FOLLOW_MACHINE.HOOK_U_IN;
        SUB1.RD_10 TO CRANE1_COME_TO_ME.HOOK_D_IN;
        SUB1.RD_10 TO CRANE1_FOLLOW_ME.HOOK_D_IN;
        SUB1.RD_10 TO CRANE1_FOLLOW_MACHINE.HOOK_D_IN;
        SUB1.RD_1 TO PERMITTER_1.E_STOP;
        START_STOP_CONTROLLER_1.FMA_O TO PERMITTER_1.N_STOP;
        SUB1.RD_7 TO CRANE1_COME_TO_ME.ACTIVATE_BRIDGE;
        SUB1.RD_7 TO CRANE1_FOLLOW_MACHINE.ACTIVATE_BRIDGE;
        SUB1.RD_7 TO CRANE1_FOLLOW_ME.ACTIVATE_BRIDGE;
      END_CONNECTIONS
    END_RESOURCE
  END_DEVICE
  DEVICE CRANE_2_DEVICCE : FORTE_PC(MGR_ID := %CRANE2_IP%:61499)
    {SET_ATTRIBUTE(Profile, HOLOBLOC)} (* device profile *)
    RESOURCE EMB_RES : EMB_RES
      FBS
        CRANE2_FOLLOW_ME : CRANE2_FOLLOW_ME;
        SUBSCRIBE_10_2 : SUBSCRIBE_10(QI := 1, ID := 239.0.0.2:61497);
        CRANE2_COME_TO_ME : CRANE2_COME_TO_ME;
        START_STOP_CONTROLLER_2 : START_STOP_CONTROLLER;
        SERVER2 : SERVER_0_6(QI := 1, ID := opc_ua[/Objects/1:CRANE2]);
        CRANE2_FOLLOW_MACHINE : CRANE2_FOLLOW_MACHINE;
        SENSORS_ACTUATORS_2 : SENSORS_ACTUATORS;
        PERMITTER_2 : PERMITTER;
      END_FBS
      EVENT_CONNECTIONS
        SUBSCRIBE_10_2.IND TO CRANE2_FOLLOW_ME.REQ;
        SUBSCRIBE_10_2.IND TO CRANE2_COME_TO_ME.REQ;
        SUBSCRIBE_10_2.INITO TO START_STOP_CONTROLLER_2.INIT;
        SUBSCRIBE_10_2.IND TO START_STOP_CONTROLLER_2.REQ;
        START_STOP_CONTROLLER_2.CNF TO CRANE2_COME_TO_ME.REQ;
        START_STOP_CONTROLLER_2.CNF TO CRANE2_FOLLOW_ME.REQ;
        SERVER2.IND TO SERVER2.RSP;
        SERVER2.INITO TO SUBSCRIBE_10_2.INIT;
        SERVER2.IND TO CRANE2_COME_TO_ME.REQ;
        SERVER2.IND TO CRANE2_FOLLOW_ME.REQ;
        SERVER2.IND TO SERVER2.RSP;
        START_STOP_CONTROLLER_2.CNF TO CRANE2_FOLLOW_MACHINE.REQ;
        SERVER2.IND TO CRANE2_FOLLOW_MACHINE.REQ;
        SUBSCRIBE_10_2.IND TO CRANE2_FOLLOW_MACHINE.REQ;
        CRANE2_COME_TO_ME.CNF TO SENSORS_ACTUATORS_2.REQ;
        CRANE2_FOLLOW_ME.CNF TO SENSORS_ACTUATORS_2.REQ;
        CRANE2_FOLLOW_MACHINE.CNF TO SENSORS_ACTUATORS_2.REQ;
        SUBSCRIBE_10_2.IND TO SENSORS_ACTUATORS_2.REQ;
        SUBSCRIBE_10_2.INITO TO SENSORS_ACTUATORS_2.INIT;
        SENSORS_ACTUATORS_2.S_A_E TO CRANE2_FOLLOW_ME.MPS_E;
        SENSORS_ACTUATORS_2.S_A_E TO CRANE2_COME_TO_ME.MPS_E;
        SENSORS_ACTUATORS_2.S_A_E TO CRANE2_FOLLOW_MACHINE.MPS_E;
        START.COLD TO SERVER2.INIT;
        START.WARM TO SERVER2.INIT;
        SENSORS_ACTUATORS_2.S_A_E TO PERMITTER_2.TRIGGER_IN;
        START_STOP_CONTROLLER_2.CNF TO PERMITTER_2.REQ;
        PERMITTER_2.TRIGGER_OUT TO CRANE2_FOLLOW_MACHINE.REQ;
      END_CONNECTIONS
      DATA_CONNECTIONS
        SUBSCRIBE_10_2.RD_1 TO CRANE2_FOLLOW_ME.E_STOP;
        SUBSCRIBE_10_2.RD_2 TO CRANE2_FOLLOW_ME.TEXT_BOX;
        SUBSCRIBE_10_2.RD_6 TO CRANE2_FOLLOW_ME.CHOOSE_CRANE;
        SUBSCRIBE_10_2.RD_8 TO CRANE2_FOLLOW_ME.ACTIVATE_TROLLEY;
        SUBSCRIBE_10_2.RD_9 TO CRANE2_FOLLOW_ME.HOOK_U_IN;
        SUBSCRIBE_10_2.RD_10 TO CRANE2_FOLLOW_ME.HOOK_D_IN;
        SUBSCRIBE_10_2.RD_1 TO CRANE2_COME_TO_ME.E_STOP;
        SUBSCRIBE_10_2.RD_2 TO CRANE2_COME_TO_ME.TEXT_BOX;
        SUBSCRIBE_10_2.RD_6 TO CRANE2_COME_TO_ME.CHOOSE_CRANE;
        SUBSCRIBE_10_2.RD_8 TO CRANE2_COME_TO_ME.ACTIVATE_TROLLEY;
        SUBSCRIBE_10_2.RD_9 TO CRANE2_COME_TO_ME.HOOK_U_IN;
        SUBSCRIBE_10_2.RD_10 TO CRANE2_COME_TO_ME.HOOK_D_IN;
        SUBSCRIBE_10_2.RD_3 TO START_STOP_CONTROLLER_2.CTM;
        SUBSCRIBE_10_2.RD_4 TO START_STOP_CONTROLLER_2.FME;
        SUBSCRIBE_10_2.RD_5 TO START_STOP_CONTROLLER_2.FMA;
        START_STOP_CONTROLLER_2.CTM_O TO CRANE2_COME_TO_ME.N_STOP;
        START_STOP_CONTROLLER_2.FME_O TO CRANE2_FOLLOW_ME.N_STOP;
        SERVER2.RD_1 TO CRANE2_COME_TO_ME.X_B_LOC;
        SERVER2.RD_2 TO CRANE2_COME_TO_ME.Y_T_LOC;
        SERVER2.RD_3 TO CRANE2_FOLLOW_ME.X_B_LOC;
        SERVER2.RD_4 TO CRANE2_FOLLOW_ME.Y_T_LOC;
        SUBSCRIBE_10_2.RD_1 TO CRANE2_FOLLOW_MACHINE.E_STOP;
        START_STOP_CONTROLLER_2.FMA_O TO CRANE2_FOLLOW_MACHINE.N_STOP;
        SERVER2.RD_5 TO CRANE2_FOLLOW_MACHINE.X_B_LOC;
        SERVER2.RD_6 TO CRANE2_FOLLOW_MACHINE.Y_T_LOC;
        SUBSCRIBE_10_2.RD_2 TO CRANE2_FOLLOW_MACHINE.TEXT_BOX;
        SUBSCRIBE_10_2.RD_6 TO CRANE2_FOLLOW_MACHINE.CHOOSE_CRANE;
        SUBSCRIBE_10_2.RD_8 TO CRANE2_FOLLOW_MACHINE.ACTIVATE_TROLLEY;
        SUBSCRIBE_10_2.RD_9 TO CRANE2_FOLLOW_MACHINE.HOOK_U_IN;
        SUBSCRIBE_10_2.RD_10 TO CRANE2_FOLLOW_MACHINE.HOOK_D_IN;
        CRANE2_COME_TO_ME.A_D_MPS TO SENSORS_ACTUATORS_2.CTM_ACTIVATE_MP;
        CRANE2_COME_TO_ME.BRIDGE_F TO SENSORS_ACTUATORS_2.CTM_BRIDGE_F_I;
        CRANE2_COME_TO_ME.BRIDGE_B TO SENSORS_ACTUATORS_2.CTM_BRIGDE_B_I;
        CRANE2_COME_TO_ME.TROLLEY_F TO SENSORS_ACTUATORS_2.CTM_TROLLEY_F_I;
        CRANE2_COME_TO_ME.TROLLEY_B TO SENSORS_ACTUATORS_2.CTM_TROLLEY_B_I;
        CRANE2_COME_TO_ME.HOOK_U TO SENSORS_ACTUATORS_2.CTM_HOOK_U_I;
        CRANE2_COME_TO_ME.HOOK_D TO SENSORS_ACTUATORS_2.CTM_HOOK_D_I;
        CRANE2_FOLLOW_ME.A_D_MPS TO SENSORS_ACTUATORS_2.FME_ACTIVATE_MP;
        CRANE2_FOLLOW_ME.BRIDGE_F TO SENSORS_ACTUATORS_2.FME_BRIDGE_F_I;
        CRANE2_FOLLOW_ME.BRIDGE_B TO SENSORS_ACTUATORS_2.FME_BRIGDE_B_I;
        CRANE2_FOLLOW_ME.TROLLEY_F TO SENSORS_ACTUATORS_2.FME_TROLLEY_F_I;
        CRANE2_FOLLOW_ME.TROLLEY_B TO SENSORS_ACTUATORS_2.FME_TROLLEY_B_I;
        CRANE2_FOLLOW_ME.HOOK_U TO SENSORS_ACTUATORS_2.FME_HOOK_U_I;
        CRANE2_FOLLOW_ME.HOOK_D TO SENSORS_ACTUATORS_2.FME_HOOK_D_I;
        CRANE2_FOLLOW_MACHINE.A_D_MPS TO SENSORS_ACTUATORS_2.FMA_ACTIVATE_MP;
        SUBSCRIBE_10_2.RD_1 TO SENSORS_ACTUATORS_2.E_STOP;
        CRANE2_FOLLOW_MACHINE.BRIDGE_F TO SENSORS_ACTUATORS_2.FMA_BRIDGE_F_I;
        CRANE2_FOLLOW_MACHINE.BRIDGE_B TO SENSORS_ACTUATORS_2.FMA_BRIGDE_B_I;
        CRANE2_FOLLOW_MACHINE.TROLLEY_F TO SENSORS_ACTUATORS_2.FMA_TROLLEY_F_I;
        CRANE2_FOLLOW_MACHINE.TROLLEY_B TO SENSORS_ACTUATORS_2.FMA_TROLLEY_B_I;
        CRANE2_FOLLOW_MACHINE.HOOK_U TO SENSORS_ACTUATORS_2.FMA_HOOK_U_I;
        CRANE2_FOLLOW_MACHINE.HOOK_D TO SENSORS_ACTUATORS_2.FMA_HOOK_D_I;
        SENSORS_ACTUATORS_2.BRIDGE_P TO CRANE2_COME_TO_ME.BRIDGE_P;
        SENSORS_ACTUATORS_2.BRIDGE_P TO CRANE2_FOLLOW_ME.BRIDGE_P;
        SENSORS_ACTUATORS_2.BRIDGE_P TO CRANE2_FOLLOW_MACHINE.BRIDGE_P;
        SENSORS_ACTUATORS_2.TROLLEY_P TO CRANE2_COME_TO_ME.TROLLEY_P;
        SENSORS_ACTUATORS_2.TROLLEY_P TO CRANE2_FOLLOW_ME.TROLLEY_P;
        SENSORS_ACTUATORS_2.TROLLEY_P TO CRANE2_FOLLOW_MACHINE.TROLLEY_P;
        SENSORS_ACTUATORS_2.HOOK_P TO CRANE2_COME_TO_ME.HOOK_P;
        SENSORS_ACTUATORS_2.HOOK_P TO CRANE2_FOLLOW_ME.HOOK_P;
        SENSORS_ACTUATORS_2.HOOK_P TO CRANE2_FOLLOW_MACHINE.HOOK_P;
        SENSORS_ACTUATORS_2.CRANE_DIS_S TO CRANE2_COME_TO_ME.CRANE_DIS_S;
        SENSORS_ACTUATORS_2.CRANE_DIS_S TO CRANE2_FOLLOW_ME.CRANE_DIS_S;
        SENSORS_ACTUATORS_2.CRANE_DIS_S TO CRANE2_FOLLOW_MACHINE.CRANE_DIS_S;
        SUBSCRIBE_10_2.RD_1 TO PERMITTER_2.E_STOP;
        START_STOP_CONTROLLER_2.FMA_O TO PERMITTER_2.N_STOP;
        SUBSCRIBE_10_2.RD_7 TO CRANE2_COME_TO_ME.ACTIVATE_BRIDGE;
        SUBSCRIBE_10_2.RD_7 TO CRANE2_FOLLOW_ME.ACTIVATE_BRIDGE;
        SUBSCRIBE_10_2.RD_7 TO CRANE2_FOLLOW_MACHINE.ACTIVATE_BRIDGE;
      END_CONNECTIONS
    END_RESOURCE
  END_DEVICE
  DEVICE FBRT_WINDOW : FBRT_WINDOW(BOUNDS := [300,300,220,400], GRID := [1,1], MGR_ID := "localhost:61505")
    {SET_ATTRIBUTE(Profile, HOLOBLOC)} (* device profile *)
    RESOURCE PANEL_RESOURCE : PANEL_RESOURCE
      FBS
        HOOK_UP_DOWN : RADIO_BOOL(QI := 1, LABEL1 := Hook Down, LABEL0 := Stop, IN := 0);
        MASTER_SLAVE : RADIO_BOOL(QI := 1, LABEL1 := Activate Bridge, LABEL0 := Stop, IN := 0);
        CHOOSE_X : RADIO_BOOL(QI := 1, LABEL1 := Choose X, LABEL0 := No, IN := 0);
        INPUT_BOX : IN_ANY(QI := 1, W := 20, TYPE := INT);
        FOLLOW_MACHINE : RADIO_BOOL(QI := 1, LABEL1 := Follow machine, LABEL0 := STOP, IN := 0);
        BOOL2BOOL : BOOL2BOOL;
        INT2INT : INT2INT;
        FOLLOW_ME : RADIO_BOOL(QI := 1, LABEL1 := Follow me, LABEL0 := STOP, IN := 0);
        ACTIVATE_HOOK : RADIO_BOOL(QI := 1, LABEL1 := Hook Up, LABEL0 := Stop, IN := 0);
        EMERGENCY_STOP : RADIO_BOOL(QI := 1, LABEL1 := Start, LABEL0 := Emergency STOP, IN := 0);
        CRANE_NR : RADIO_BOOL(QI := 1, LABEL1 := Select Crane Nr, LABEL0 := No, IN := 0);
        BOOL2BOOL_1 : BOOL2BOOL;
        CHOOSE_Y : RADIO_BOOL(QI := 1, LABEL1 := Choose Y, LABEL0 := No, IN := 0);
        ACTIVATE_TROLLEY : RADIO_BOOL(QI := 1, LABEL1 := Activate Trolley, LABEL0 := Stop, IN := 0);
        COME_TO_ME : RADIO_BOOL(QI := 1, LABEL1 := Come to me, LABEL0 := STOP, IN := 0);
        PUBLISH_12 : PUBLISH_12(QI := 1, ID := 239.0.0.1:61496);
      END_FBS
      EVENT_CONNECTIONS
        HOOK_UP_DOWN.INITO TO CHOOSE_X.INIT;
        CHOOSE_X.IND TO BOOL2BOOL.REQ;
        INPUT_BOX.IND TO INT2INT.REQ;
        FOLLOW_ME.INITO TO FOLLOW_MACHINE.INIT;
        ACTIVATE_HOOK.INITO TO HOOK_UP_DOWN.INIT;
        EMERGENCY_STOP.INITO TO INPUT_BOX.INIT;
        FOLLOW_MACHINE.INITO TO CRANE_NR.INIT;
        CRANE_NR.INITO TO MASTER_SLAVE.INIT;
        CHOOSE_X.INITO TO CHOOSE_Y.INIT;
        CHOOSE_Y.IND TO BOOL2BOOL_1.REQ;
        MASTER_SLAVE.INITO TO ACTIVATE_TROLLEY.INIT;
        ACTIVATE_TROLLEY.INITO TO ACTIVATE_HOOK.INIT;
        INPUT_BOX.INITO TO COME_TO_ME.INIT;
        COME_TO_ME.INITO TO FOLLOW_ME.INIT;
        PUBLISH_12.INITO TO EMERGENCY_STOP.INIT;
        EMERGENCY_STOP.IND TO PUBLISH_12.REQ;
        INT2INT.CNF TO PUBLISH_12.REQ;
        COME_TO_ME.IND TO PUBLISH_12.REQ;
        FOLLOW_ME.IND TO PUBLISH_12.REQ;
        FOLLOW_MACHINE.IND TO PUBLISH_12.REQ;
        CRANE_NR.IND TO PUBLISH_12.REQ;
        MASTER_SLAVE.IND TO PUBLISH_12.REQ;
        ACTIVATE_TROLLEY.IND TO PUBLISH_12.REQ;
        ACTIVATE_HOOK.IND TO PUBLISH_12.REQ;
        HOOK_UP_DOWN.IND TO PUBLISH_12.REQ;
        BOOL2BOOL.CNF TO PUBLISH_12.REQ;
        BOOL2BOOL_1.CNF TO PUBLISH_12.REQ;
        START.COLD TO PUBLISH_12.INIT;
        START.WARM TO PUBLISH_12.INIT;
      END_CONNECTIONS
      DATA_CONNECTIONS
        CHOOSE_X.OUT TO BOOL2BOOL.IN;
        INPUT_BOX.OUT TO INT2INT.IN;
        CHOOSE_Y.OUT TO BOOL2BOOL_1.IN;
        EMERGENCY_STOP.OUT TO PUBLISH_12.SD_1;
        INT2INT.OUT TO PUBLISH_12.SD_2;
        COME_TO_ME.OUT TO PUBLISH_12.SD_3;
        FOLLOW_ME.OUT TO PUBLISH_12.SD_4;
        FOLLOW_MACHINE.OUT TO PUBLISH_12.SD_5;
        CRANE_NR.OUT TO PUBLISH_12.SD_6;
        MASTER_SLAVE.OUT TO PUBLISH_12.SD_7;
        ACTIVATE_TROLLEY.OUT TO PUBLISH_12.SD_8;
        ACTIVATE_HOOK.OUT TO PUBLISH_12.SD_9;
        HOOK_UP_DOWN.OUT TO PUBLISH_12.SD_10;
        BOOL2BOOL.OUT TO PUBLISH_12.SD_11;
        BOOL2BOOL_1.OUT TO PUBLISH_12.SD_12;
      END_CONNECTIONS
    END_RESOURCE
  END_DEVICE
  MAPPINGS
    Distributed_Control_System_OPCUA_4DiacApp.HMI_FOLLOW_ME ON HMI_DEVICE.EMB_RES.HMI_FOLLOW_ME;
    Distributed_Control_System_OPCUA_4DiacApp.HMI_COME_TO_ME ON HMI_DEVICE.EMB_RES.HMI_COME_TO_ME;
    Distributed_Control_System_OPCUA_4DiacApp.TYPE_CONVERTER ON HMI_DEVICE.EMB_RES.TYPE_CONVERTER;
    Distributed_Control_System_OPCUA_4DiacApp.FUNCTIONALITY_CONTROLLER ON HMI_DEVICE.EMB_RES.FUNCTIONALITY_CONTROLLER;
    Distributed_Control_System_OPCUA_4DiacApp.HMI_FOLLOW_MACHINE ON HMI_DEVICE.EMB_RES.HMI_FOLLOW_MACHINE;
    Distributed_Control_System_OPCUA_4DiacApp.HOOK_UP_DOWN ON FBRT_WINDOW.PANEL_RESOURCE.HOOK_UP_DOWN;
    Distributed_Control_System_OPCUA_4DiacApp.MASTER_SLAVE ON FBRT_WINDOW.PANEL_RESOURCE.MASTER_SLAVE;
    Distributed_Control_System_OPCUA_4DiacApp.CHOOSE_X ON FBRT_WINDOW.PANEL_RESOURCE.CHOOSE_X;
    Distributed_Control_System_OPCUA_4DiacApp.INPUT_BOX ON FBRT_WINDOW.PANEL_RESOURCE.INPUT_BOX;
    Distributed_Control_System_OPCUA_4DiacApp.FOLLOW_MACHINE ON FBRT_WINDOW.PANEL_RESOURCE.FOLLOW_MACHINE;
    Distributed_Control_System_OPCUA_4DiacApp.BOOL2BOOL ON FBRT_WINDOW.PANEL_RESOURCE.BOOL2BOOL;
    Distributed_Control_System_OPCUA_4DiacApp.INT2INT ON FBRT_WINDOW.PANEL_RESOURCE.INT2INT;
    Distributed_Control_System_OPCUA_4DiacApp.FOLLOW_ME ON FBRT_WINDOW.PANEL_RESOURCE.FOLLOW_ME;
    Distributed_Control_System_OPCUA_4DiacApp.ACTIVATE_HOOK ON FBRT_WINDOW.PANEL_RESOURCE.ACTIVATE_HOOK;
    Distributed_Control_System_OPCUA_4DiacApp.EMERGENCY_STOP ON FBRT_WINDOW.PANEL_RESOURCE.EMERGENCY_STOP;
    Distributed_Control_System_OPCUA_4DiacApp.CRANE_NR ON FBRT_WINDOW.PANEL_RESOURCE.CRANE_NR;
    Distributed_Control_System_OPCUA_4DiacApp.BOOL2BOOL_1 ON FBRT_WINDOW.PANEL_RESOURCE.BOOL2BOOL_1;
    Distributed_Control_System_OPCUA_4DiacApp.CHOOSE_Y ON FBRT_WINDOW.PANEL_RESOURCE.CHOOSE_Y;
    Distributed_Control_System_OPCUA_4DiacApp.ACTIVATE_TROLLEY ON FBRT_WINDOW.PANEL_RESOURCE.ACTIVATE_TROLLEY;
    Distributed_Control_System_OPCUA_4DiacApp.COME_TO_ME ON FBRT_WINDOW.PANEL_RESOURCE.COME_TO_ME;
    Distributed_Control_System_OPCUA_4DiacApp.CRANE_1 ON HMI_DEVICE.EMB_RES.CRANE_1;
    Distributed_Control_System_OPCUA_4DiacApp.CEANE_2 ON HMI_DEVICE.EMB_RES.CEANE_2;
    Distributed_Control_System_OPCUA_4DiacApp.CRANE_SELECTOR ON HMI_DEVICE.EMB_RES.CRANE_SELECTOR;
    Distributed_Control_System_OPCUA_4DiacApp.FME_FMA_DECIDER ON HMI_DEVICE.EMB_RES.FME_FMA_DECIDER;
    Distributed_Control_System_OPCUA_4DiacApp.PUBLISH_10 ON HMI_DEVICE.EMB_RES.PUBLISH_10;
    Distributed_Control_System_OPCUA_4DiacApp.PUBLISH_12 ON FBRT_WINDOW.PANEL_RESOURCE.PUBLISH_12;
    Distributed_Control_System_OPCUA_4DiacApp.SUBSCRIBE_12 ON HMI_DEVICE.EMB_RES.SUBSCRIBE_12;
    Distributed_Control_System_OPCUA_4DiacApp.CRANE2_FOLLOW_ME ON CRANE_2_DEVICCE.EMB_RES.CRANE2_FOLLOW_ME;
    Distributed_Control_System_OPCUA_4DiacApp.SUBSCRIBE_10_2 ON CRANE_2_DEVICCE.EMB_RES.SUBSCRIBE_10_2;
    Distributed_Control_System_OPCUA_4DiacApp.CRANE2_COME_TO_ME ON CRANE_2_DEVICCE.EMB_RES.CRANE2_COME_TO_ME;
    Distributed_Control_System_OPCUA_4DiacApp.START_STOP_CONTROLLER_2 ON CRANE_2_DEVICCE.EMB_RES.START_STOP_CONTROLLER_2;
    Distributed_Control_System_OPCUA_4DiacApp.SERVER2 ON CRANE_2_DEVICCE.EMB_RES.SERVER2;
    Distributed_Control_System_OPCUA_4DiacApp.CRANE2_FOLLOW_MACHINE ON CRANE_2_DEVICCE.EMB_RES.CRANE2_FOLLOW_MACHINE;
    Distributed_Control_System_OPCUA_4DiacApp.SENSORS_ACTUATORS_2 ON CRANE_2_DEVICCE.EMB_RES.SENSORS_ACTUATORS_2;
    Distributed_Control_System_OPCUA_4DiacApp.CRANE1_COME_TO_ME ON CRANE_1_DEVICCE.EMB_RES.CRANE1_COME_TO_ME;
    Distributed_Control_System_OPCUA_4DiacApp.CRANE1_FOLLOW_MACHINE ON CRANE_1_DEVICCE.EMB_RES.CRANE1_FOLLOW_MACHINE;
    Distributed_Control_System_OPCUA_4DiacApp.CRANE1_FOLLOW_ME ON CRANE_1_DEVICCE.EMB_RES.CRANE1_FOLLOW_ME;
    Distributed_Control_System_OPCUA_4DiacApp.SERVER1 ON CRANE_1_DEVICCE.EMB_RES.SERVER1;
    Distributed_Control_System_OPCUA_4DiacApp.START_STOP_CONTROLLER_1 ON CRANE_1_DEVICCE.EMB_RES.START_STOP_CONTROLLER_1;
    Distributed_Control_System_OPCUA_4DiacApp.SENSORS_ACTUATORS_1 ON CRANE_1_DEVICCE.EMB_RES.SENSORS_ACTUATORS_1;
    Distributed_Control_System_OPCUA_4DiacApp.SUB1 ON CRANE_1_DEVICCE.EMB_RES.SUB1;
    Distributed_Control_System_OPCUA_4DiacApp.REQUEST ON HMI_DEVICE.EMB_RES.REQUEST;
    Distributed_Control_System_OPCUA_4DiacApp.RESPONSE ON HMI_DEVICE.EMB_RES.RESPONSE;
    Distributed_Control_System_OPCUA_4DiacApp.PERMITTER_1 ON CRANE_1_DEVICCE.EMB_RES.PERMITTER_1;
    Distributed_Control_System_OPCUA_4DiacApp.PERMITTER_2 ON CRANE_2_DEVICCE.EMB_RES.PERMITTER_2;
  END_MAPPINGS
  SEGMENTS
    Ethernet : Ethernet;
  END_SEGMENTS
  LINKS
    FBRT_WINDOW => Ethernet;
    HMI_DEVICE => Ethernet;
    CRANE_1_DEVICCE => Ethernet;
    CRANE_2_DEVICCE => Ethernet;
  END_LINKS
END_SYSTEM
